(*
    Evaluates all interlock conditions (HV, calibration, reference, sensor) in both directions for RET, X, Y, and Z axes.
    Outputs bSafeToMove* flags for each axis and overall, enabling sequence or maintenance moves only when all safety criteria are met.
*)
FUNCTION_BLOCK  FB_DGPDEPS
VAR_IN_OUT
    stMotionStageRET : ST_MotionStage;
    stMotionStageX	 : ST_MotionStage;
    stMotionStageY   : ST_MotionStage;
    stMotionStageZ   : ST_MotionStage;
	
    stMCS2ChanParameterRET : ST_MCS2ChanParameter;
    stMCS2ChanParameterX   : ST_MCS2ChanParameter;
    stMCS2ChanParameterY   : ST_MCS2ChanParameter;
    stMCS2ChanParameterZ   : ST_MCS2ChanParameter;
END_VAR

VAR_INPUT
    bHVActive : BOOL;
    bEnable   : BOOL := TRUE;
END_VAR

VAR_OUTPUT
    bSafeToMoveRET : BOOL;
    bSafeToMoveX   : BOOL;
    bSafeToMoveY   : BOOL;
    bSafeToMoveZ   : BOOL;
    bSafeToMove    : BOOL;
END_VAR

VAR
    // RET
    epsHVRETPositive, epsHVRETNegative       : FB_EPS;
    epsCalRETPositive, epsCalRETNegative     : FB_EPS;
    epsRefRETPositive, epsRefRETNegative     : FB_EPS;
    epsSensRETPositive, epsSensRETNegative   : FB_EPS;
    // X
    epsHVXPositive, epsHVXNegative           : FB_EPS;
    epsCalXPositive, epsCalXNegative         : FB_EPS;
    epsRefXPositive, epsRefXNegative         : FB_EPS;
    epsSensXPositive, epsSensXNegative       : FB_EPS;
    // Y
    epsHVYPositive, epsHVYNegative           : FB_EPS;
    epsCalYPositive, epsCalYNegative         : FB_EPS;
    epsRefYPositive, epsRefYNegative         : FB_EPS;
    epsSensYPositive, epsSensYNegative       : FB_EPS;
    // Z
    epsHVZPositive, epsHVZNegative           : FB_EPS;
    epsCalZPositive, epsCalZNegative         : FB_EPS;
    epsRefZPositive, epsRefZNegative         : FB_EPS;
    epsSensZPositive, epsSensZNegative       : FB_EPS;
END_VAR

IF NOT __ISVALIDREF(stMotionStageRET)
    OR NOT __ISVALIDREF(stMotionStageX)
    OR NOT __ISVALIDREF(stMotionStageY)
    OR NOT __ISVALIDREF(stMotionStageZ)
	OR NOT __ISVALIDREF(stMCS2ChanParameterRET)
    OR NOT __ISVALIDREF(stMCS2ChanParameterX)
    OR NOT __ISVALIDREF(stMCS2ChanParameterY)
    OR NOT __ISVALIDREF(stMCS2ChanParameterZ)
THEN
    RETURN;
END_IF

IF bEnable THEN
    // =========== RET EPS Directional Checks ===========
    epsHVRETPositive(eps := stMotionStageRET.stEPSForwardEnable);
    epsHVRETPositive.setBit(nBits := 0, bValue := NOT bHVActive);
    epsCalRETPositive(eps := stMotionStageRET.stEPSForwardEnable);
    epsCalRETPositive.setBit(nBits := 1, bValue := stMCS2ChanParameterRET.stChannelState.bIsCalibrated);
    epsRefRETPositive(eps := stMotionStageRET.stEPSForwardEnable);
    epsRefRETPositive.setBit(nBits := 2, bValue := stMCS2ChanParameterRET.stChannelState.bIsReferenced);
    epsSensRETPositive(eps := stMotionStageRET.stEPSForwardEnable);
    epsSensRETPositive.setBit(nBits := 3, bValue := stMCS2ChanParameterRET.stChannelState.bSensorPresent);

    epsHVRETNegative(eps := stMotionStageRET.stEPSBackwardEnable);
    epsHVRETNegative.setBit(nBits := 0, bValue := NOT bHVActive);
    epsCalRETNegative(eps := stMotionStageRET.stEPSBackwardEnable);
    epsCalRETNegative.setBit(nBits := 1, bValue := stMCS2ChanParameterRET.stChannelState.bIsCalibrated);
    epsRefRETNegative(eps := stMotionStageRET.stEPSBackwardEnable);
    epsRefRETNegative.setBit(nBits := 2, bValue := stMCS2ChanParameterRET.stChannelState.bIsReferenced);
    epsSensRETNegative(eps := stMotionStageRET.stEPSBackwardEnable);
    epsSensRETNegative.setBit(nBits := 3, bValue := stMCS2ChanParameterRET.stChannelState.bSensorPresent);

    bSafeToMoveRET :=
        stMotionStageRET.stEPSForwardEnable.bEPS_OK
        AND stMotionStageRET.stEPSBackwardEnable.bEPS_OK;

    // =========== X Axis EPS Directional Checks ===========
    epsHVXPositive(eps := stMotionStageX.stEPSForwardEnable);
    epsHVXPositive.setBit(nBits := 0, bValue := NOT bHVActive);
    epsCalXPositive(eps := stMotionStageX.stEPSForwardEnable);
    epsCalXPositive.setBit(nBits := 1, bValue := stMCS2ChanParameterX.stChannelState.bIsCalibrated);
    epsRefXPositive(eps := stMotionStageX.stEPSForwardEnable);
    epsRefXPositive.setBit(nBits := 2, bValue := stMCS2ChanParameterX.stChannelState.bIsReferenced);
    epsSensXPositive(eps := stMotionStageX.stEPSForwardEnable);
    epsSensXPositive.setBit(nBits := 3, bValue := stMCS2ChanParameterX.stChannelState.bSensorPresent);

    epsHVXNegative(eps := stMotionStageX.stEPSBackwardEnable);
    epsHVXNegative.setBit(nBits := 0, bValue := NOT bHVActive);
    epsCalXNegative(eps := stMotionStageX.stEPSBackwardEnable);
    epsCalXNegative.setBit(nBits := 1, bValue := stMCS2ChanParameterX.stChannelState.bIsCalibrated);
    epsRefXNegative(eps := stMotionStageX.stEPSBackwardEnable);
    epsRefXNegative.setBit(nBits := 2, bValue := stMCS2ChanParameterX.stChannelState.bIsReferenced);
    epsSensXNegative(eps := stMotionStageX.stEPSBackwardEnable);
    epsSensXNegative.setBit(nBits := 3, bValue := stMCS2ChanParameterX.stChannelState.bSensorPresent);

    bSafeToMoveX :=
        stMotionStageX.stEPSForwardEnable.bEPS_OK
        AND stMotionStageX.stEPSBackwardEnable.bEPS_OK;

    // =========== Y Axis EPS Directional Checks ===========
    epsHVYPositive(eps := stMotionStageY.stEPSForwardEnable);
    epsHVYPositive.setBit(nBits := 0, bValue := NOT bHVActive);
    epsCalYPositive(eps := stMotionStageY.stEPSForwardEnable);
    epsCalYPositive.setBit(nBits := 1, bValue := stMCS2ChanParameterY.stChannelState.bIsCalibrated);
    epsRefYPositive(eps := stMotionStageY.stEPSForwardEnable);
    epsRefYPositive.setBit(nBits := 2, bValue := stMCS2ChanParameterY.stChannelState.bIsReferenced);
    epsSensYPositive(eps := stMotionStageY.stEPSForwardEnable);
    epsSensYPositive.setBit(nBits := 3, bValue := stMCS2ChanParameterY.stChannelState.bSensorPresent);

    epsHVYNegative(eps := stMotionStageY.stEPSBackwardEnable);
    epsHVYNegative.setBit(nBits := 0, bValue := NOT bHVActive);
    epsCalYNegative(eps := stMotionStageY.stEPSBackwardEnable);
    epsCalYNegative.setBit(nBits := 1, bValue := stMCS2ChanParameterY.stChannelState.bIsCalibrated);
    epsRefYNegative(eps := stMotionStageY.stEPSBackwardEnable);
    epsRefYNegative.setBit(nBits := 2, bValue := stMCS2ChanParameterY.stChannelState.bIsReferenced);
    epsSensYNegative(eps := stMotionStageY.stEPSBackwardEnable);
    epsSensYNegative.setBit(nBits := 3, bValue := stMCS2ChanParameterY.stChannelState.bSensorPresent);

    bSafeToMoveY :=
        stMotionStageY.stEPSForwardEnable.bEPS_OK
        AND stMotionStageY.stEPSBackwardEnable.bEPS_OK;

    // =========== Z Axis EPS Directional Checks ===========
    epsHVZPositive(eps := stMotionStageZ.stEPSForwardEnable);
    epsHVZPositive.setBit(nBits := 0, bValue := NOT bHVActive);
    epsCalZPositive(eps := stMotionStageZ.stEPSForwardEnable);
    epsCalZPositive.setBit(nBits := 1, bValue := stMCS2ChanParameterZ.stChannelState.bIsCalibrated);
    epsRefZPositive(eps := stMotionStageZ.stEPSForwardEnable);
    epsRefZPositive.setBit(nBits := 2, bValue := stMCS2ChanParameterZ.stChannelState.bIsReferenced);
    epsSensZPositive(eps := stMotionStageZ.stEPSForwardEnable);
    epsSensZPositive.setBit(nBits := 3, bValue :=stMCS2ChanParameterZ.stChannelState.bSensorPresent);

    epsHVZNegative(eps := stMotionStageZ.stEPSBackwardEnable);
    epsHVZNegative.setBit(nBits := 0, bValue := NOT bHVActive);
    epsCalZNegative(eps := stMotionStageZ.stEPSBackwardEnable);
    epsCalZNegative.setBit(nBits := 1, bValue := stMCS2ChanParameterZ.stChannelState.bIsCalibrated);
    epsRefZNegative(eps := stMotionStageZ.stEPSBackwardEnable);
    epsRefZNegative.setBit(nBits := 2, bValue := stMCS2ChanParameterZ.stChannelState.bIsReferenced);
    epsSensZNegative(eps := stMotionStageZ.stEPSBackwardEnable);
    epsSensZNegative.setBit(nBits := 3, bValue := stMCS2ChanParameterZ.stChannelState.bSensorPresent);

    bSafeToMoveZ :=
        stMotionStageZ.stEPSForwardEnable.bEPS_OK
        AND stMotionStageZ.stEPSBackwardEnable.bEPS_OK;

    // --- Global output ---
    bSafeToMove := bSafeToMoveRET AND bSafeToMoveX AND bSafeToMoveY AND bSafeToMoveZ;
END_IF

(*
    Evaluates the RET interlocks in maintenance mode, combining the positive and negative EPS directions,
    to permit RET movement only if bRETSafeToMove is TRUE.
    This method is called exclusively during maintenance mode to ensure safe, interlocked RET axis operation.
*)
METHOD epsMaintenanceMode : BOOL
VAR_INST
//     epsSafetToMoveRETPositive  : FB_EPS;
//     epsSafetToMoveRETNegative  : FB_EPS;
	epsSafetToMoveRET  : FB_EPS;
END_VAR

VAR_INPUT
    bRETSafeToMove : BOOL;
END_VAR
IF bEnable THEN
    epsSafetToMoveRET(eps := stMotionStageRET.stEPSPowerEnable);
    epsSafetToMoveRET.setBit(nBits := 1, bValue := bRETSafeToMove);
	IF NOT bRETSafeToMove THEN
		stMotionStageRET.sCustomErrorMessage := 'RET Locked out: Address collision avoidance hazard';
	END_IF
END_IF
END_METHOD

END_FUNCTION_BLOCK

(* stored: Version 1.1.0.1
   POU FB_DGPDEPS: Id {e129cc81-4ab3-4137-8196-cf610077894e}, SpecialFunc None
   Method epsMaintenanceMode: Id {05d29efd-64cb-4db9-9e5f-5126034d60b6} *)
